FUNCTION_BLOCK FB_StationT2
VAR_IN_OUT
	XpMover			: MC_PlanarMover;
	XpTrack			: ARRAY [*] OF MC_PlanarTrack;
END_VAR
VAR_INPUT
	execute			: BOOL;
	bT3Occupied		: BOOL;
	bT3BeforeRotate	: BOOL;
END_VAR
VAR_OUTPUT
	bOccupied		: BOOL;
	bReady			: BOOL;
	bDone			: BOOL;
END_VAR
VAR
	nState			: INT;
	fbMoveTrack		: FB_XpMoveTrack;
	fbMoveC			: FB_XpMoveC;
	nTargetTrack	: INT;
	bMove			: BOOL;
	bMoveC			: BOOL;
	nRotatePos		: LREAL :=0;
END_VAR

CASE nState OF
	0: //init
	IF execute THEN
		bOccupied := TRUE;//Stationの状態をOccupiedにする
		bReady	:= FALSE;
		nState := 10;
	END_IF
	
	10://T3のMover待ち
	IF bT3Occupied THEN
		bDone := FALSE;
		nState := 20;
	END_IF
	
	
	20://移動
	ntargetTrack:= E_TrackName.T2_2_ToRotate;
	fbMoveTrack.execute:= TRUE;
	
	IF fbMoveTrack.done THEN
		fbMoveTrack.execute:= FALSE;
		bOccupied := FALSE;
		bReady := TRUE;//Stationの状態をREADYにする
		nState := 30;
	END_IF
	
	30://回転
	IF bT3BeforeRotate THEN //T3のMoverが到着したら
		fbMoveC.execute:= TRUE;
	END_IF
	IF fbMoveC.done THEN
		fbMoveC.execute := FALSE;
		nState := 40;
	END_IF
	
	40:	//T1へ移動
	nTargetTrack := E_TrackName.T1_1_ToRotate;
	fbMoveTrack.execute:= TRUE;
	bOccupied := FALSE;
	nState := 50;
	
	50:
	IF fbMoveTrack.done THEN
		fbMoveTrack.execute := FALSE;//移動指令を落とす
		bReady :=TRUE;
		bDone :=TRUE;
		nState := 100;
	END_IF

	100://initへ戻る
	nState := 0;
END_CASE

//IF bMove THEN
	fbMoveTrack(XpMover:= XpMover, 
				XpTrack:= XpTrack[nTargetTrack]);
//ELSIF bMoveC THEN	
	fbMoveC(XpMover:= XpMover, 
			position:= nRotatePos + 360);
//END_IF

END_FUNCTION_BLOCK

(* stored: Version 1.1.0.1
   POU FB_StationT2: Id {e2265522-30f6-430e-aa61-2d3bf796ce24}, SpecialFunc None *)
